TYPE "Rework_ShW"
VERSION : 0.1
   STRUCT
      Trigger : Bool;
      Result : Int;
      Completed : Bool;
   END_STRUCT;

END_TYPE

